(* IEC 61131-3 sources: rules_plc/examples/simple_3, 3 files *)

(* ---- can_types.dut ---- *)
TYPE CAN_MSG_BUFFER :
STRUCT
	dwStart : DWORD;
	byte1 : USINT;
	byte2 : USINT;
	byte3 : USINT;
	byte4 : USINT;
	byte5 : USINT;
	byte6 : USINT;
	byte7 : USINT;
	byte8 : USINT;
	bEnd : BYTE;
END_STRUCT;
END_TYPE

TYPE CAN_MSG :
STRUCT
   value_byte: USINT;
END_STRUCT;
END_TYPE

(* ---- can_reader.st ---- *)
FUNCTION_BLOCK CAN_READER
    VAR
        buffer: CAN_MSG_BUFFER;
    END_VAR
    VAR_IN_OUT
        out_msg: CAN_MSG;
    END_VAR

    buffer.byte1 := buffer.byte1 + 1;

    out_msg.value_byte := buffer.byte1;

END_FUNCTION_BLOCK

(* ---- main_program.st ---- *)
PROGRAM main_program
    VAR
        result : CAN_MSG;
        reader_fb: CAN_READER;
    END_VAR

    reader_fb(out_msg := result);
    reader_fb(out_msg := result);

END_PROGRAM
